// TwinCAT 3 PLC project Cycler
// ProgramVersion: 3.1.4020.4
// libraries:
//   Tc2_Drive, * (Beckhoff Automation GmbH)
//   Tc2_MC2, * (Beckhoff Automation GmbH)
//   Tc2_MC2_Drive, * (Beckhoff Automation GmbH)
//   Tc2_NcDrive, * (Beckhoff Automation GmbH)
//   Tc2_Standard, * (Beckhoff Automation GmbH)
//   Tc2_System, * (Beckhoff Automation GmbH)
//   Tc3_MC2_AdvancedHoming, * (Beckhoff Automation GmbH)
//   Tc3_Module, * (Beckhoff Automation GmbH)
//   VisuDialogs, * (System)
// project tree:
//   DUTs/ AxisInfo.TcDUT, ShutterSide.TcDUT, ShutterState.TcDUT
//   / GlobalTextList.TcGTLO, PlcTask.TcTTO, Visualization Manager.TcVMO (not stored)
//   GVLs/ GVL.TcGVL
//   POUs/ Cycler.TcPOU, TestMotion.TcPOU, MAIN.TcPOU
//   VISUs/ CyclerGUI.TcVIS, TestMotionGUI.TcVIS
// real-time tasks:
//   TASK PlcTask: cycle T#1ms, priority 20, ADS port 350
// motion (NC):
//   TASK NC-Task 1 SAF: cycle T#1ms, priority 4, ADS port 501
//   TASK NC-Task 1 SVB: cycle T#10ms, priority 8, ADS port 511
//   AXIS Axis 1 (id 1)
//     Dynamic: Acceleration=7407.41, Deceleration=7407.41, Jerk=32921.8
//     Velo: RefSearch=60, SlowManual=150
//     OtherSettings: AllowMotionCmdToSlave=true
//     encoder EncType=4
//       EncPara: ScaleFactorNumerator=0.049777676567, MaxCount=#x0000ffff
//         SoftEndMaxControl: Range=749
//         Inc: RefSearchInverse=true, RefSyncInverse=false, RefSoftSyncMask=#x0000ffff
//         TimeComp: TimeCompMode=1, EncDelayCycles=4
//     drive DrvType=24
//       Analog: VeloReferenz=2038.894
//       TimeComp: TaskDelayCycles=1
//     controller CtrType=1
//       CtrPara: PriorControlFactor=1
//         PosDiffControl: Range=2.5, Time=0.01
//         Observer: BandWidth=20
//   AXIS Axis 2 (id 2)
//     Dynamic: Acceleration=7407.41, Deceleration=7407.41, Jerk=32921.8
//     Velo: RefSearch=60
//     OtherSettings: AllowMotionCmdToSlave=true
//     encoder EncType=4
//       EncPara: ScaleFactorNumerator=0.049777676567, MaxCount=#x0000ffff
//         SoftEndMaxControl: Range=749
//         Inc: RefSoftSyncMask=#x0000ffff
//         TimeComp: TimeCompMode=1, EncDelayCycles=4
//     drive DrvType=24
//       Analog: VeloReferenz=2038.894
//       TimeComp: TaskDelayCycles=1
//     controller CtrType=1
//       CtrPara: PriorControlFactor=1
//         PosDiffControl: Range=2.5, Time=0.01
//         Observer: BandWidth=20
// I/O:
//   DEVICE Device 1 (EtherCAT), AmsNetId 5.48.66.18.2.1
//     Term 1 (EK1200) [EK1200-5000 EtherCAT Power supply (2A E-Bus)]
//       Term 2 (EL7047) [EL7047 1Ch. Stepper motor output stage (50V, 5A)]
//       Term 3 (EL1819) [EL1819 16Ch. Dig. Input 24V, 10µs]
//       Term 9 (EL1258) [EL1258 8Ch. Dig Input 24V with Multi-Time-Stamp]
//       Term 10 (EL1259) [EL1259 8Ch. Dig Input 24V/8Ch. Dig. Output 24V with Multi-Time-Stamp]
//       Term 4 (EL7047) [EL7047 1Ch. Stepper motor output stage (50V, 5A)]
//       Term 5 (EL2622) [EL2622 2Ch. Relay Output, NO (230V AC / 30V DC)]
//       Term 14 (EK1110) [EK1110 EtherCAT extension]
//     Term 15 (EK1100) [EK1100 EtherCAT Coupler (2A E-Bus)]
//       Term 16 (EL3681) [EL3681 Digital multimeter terminal]
//       Term 17 (EL3318) [EL3318 8Ch. Ana Input Thermocouple (TC)]
//       Term 23 (EL9011) [EL9011 End Terminal]
//     Term 18 (EK1100) [EK1100 EtherCAT Coupler (2A E-Bus)]
//       Term 19 (EL3602) [EL3602 2Ch. Ana. Input +/-10Volt, Diff. 24bit]
//       Term 20 (EL3602) [EL3602 2Ch. Ana. Input +/-10Volt, Diff. 24bit]
//       Term 24 (EL9011) [EL9011 End Terminal]
// variable links:
//   (this object) <-> Device 1 (EtherCAT)/Term 1 (EK1200)/Term 2 (EL7047)
//     Drive/Inputs/In/nState1 @bit 3 <-> STM Status/Status/Error
//     Drive/Inputs/In/nState1 @bit 7 <-> STM Status/Status/Motor stall
//     Drive/Inputs/In/nState1 @bit 5 <-> STM Status/Status/Moving negative
//     Drive/Inputs/In/nState1 @bit 4 <-> STM Status/Status/Moving positive
//     Drive/Inputs/In/nState1 @bit 1 <-> STM Status/Status/Ready
//     Drive/Inputs/In/nState1 <-> STM Status/Status/Ready to enable
//     Drive/Inputs/In/nState1 @bit 6 <-> STM Status/Status/Torque reduced
//     Drive/Inputs/In/nState1 @bit 2 <-> STM Status/Status/Warning
//     Drive/Inputs/In/nState2 @bit 4 <-> STM Status/Status/Digital input 2
//     Drive/Inputs/In/nState2 @bit 5 <-> STM Status/Status/Sync error
//     Drive/Inputs/In/nState2 @bit 7 <-> STM Status/Status/TxPDO Toggle
//     Drive/Inputs/In/nState4 @bit 1 <-> WcState/InputToggle
//     Drive/Inputs/In/nState4 <-> WcState/WcState
//     Drive/Outputs/Out/nCtrl1 <-> STM Control/Control/Enable
//     Drive/Outputs/Out/nCtrl1 @bit 2 <-> STM Control/Control/Reduce torque
//     Drive/Outputs/Out/nCtrl1 @bit 1 <-> STM Control/Control/Reset
//     Drive/Outputs/Out/nCtrl2 @bit 3 <-> STM Control/Control/Digital output 1
//     Drive/Outputs/Out/nDataOut2[0] <-> STM Velocity/Velocity
//     Enc/Inputs/In/nDataIn1[0] <-> ENC Status compact/Counter value
//     Enc/Inputs/In/nDataIn2[0] <-> ENC Status compact/Latch value
//     Enc/Inputs/In/nState1 @bit 4 <-> ENC Status compact/Status/Counter overflow
//     Enc/Inputs/In/nState1 @bit 3 <-> ENC Status compact/Status/Counter underflow
//     Enc/Inputs/In/nState1 @bit 7 <-> ENC Status compact/Status/Extrapolation stall
//     Enc/Inputs/In/nState1 <-> ENC Status compact/Status/Latch C valid
//     Enc/Inputs/In/nState1 @bit 1 <-> ENC Status compact/Status/Latch extern valid
//     Enc/Inputs/In/nState1 @bit 2 <-> ENC Status compact/Status/Set counter done
//     Enc/Inputs/In/nState2 @bit 4 <-> ENC Status compact/Status/Status of extern latch
//     Enc/Inputs/In/nState2 <-> ENC Status compact/Status/Status of input A
//     Enc/Inputs/In/nState2 @bit 1 <-> ENC Status compact/Status/Status of input B
//     Enc/Inputs/In/nState2 @bit 2 <-> ENC Status compact/Status/Status of input C
//     Enc/Inputs/In/nState2 @bit 5 <-> ENC Status compact/Status/Sync error
//     Enc/Inputs/In/nState2 @bit 7 <-> ENC Status compact/Status/TxPDO Toggle
//     Enc/Inputs/In/nState4 @bit 1 <-> WcState/InputToggle
//     Enc/Inputs/In/nState4 <-> WcState/WcState
//     Enc/Outputs/Out/nCtrl1 <-> ENC Control compact/Control/Enable latch C
//     Enc/Outputs/Out/nCtrl1 @bit 3 <-> ENC Control compact/Control/Enable latch extern on negative edge
//     Enc/Outputs/Out/nCtrl1 @bit 1 <-> ENC Control compact/Control/Enable latch extern on positive edge
//     Enc/Outputs/Out/nCtrl1 @bit 2 <-> ENC Control compact/Control/Set counter
//     Enc/Outputs/Out/nDataOut1[0] <-> ENC Control compact/Set counter value
//   (this object) <-> Device 1 (EtherCAT)/Term 1 (EK1200)/Term 4 (EL7047)
//     Drive/Inputs/In/nState1 @bit 3 <-> STM Status/Status/Error
//     Drive/Inputs/In/nState1 @bit 7 <-> STM Status/Status/Motor stall
//     Drive/Inputs/In/nState1 @bit 5 <-> STM Status/Status/Moving negative
//     Drive/Inputs/In/nState1 @bit 4 <-> STM Status/Status/Moving positive
//     Drive/Inputs/In/nState1 @bit 1 <-> STM Status/Status/Ready
//     Drive/Inputs/In/nState1 <-> STM Status/Status/Ready to enable
//     Drive/Inputs/In/nState1 @bit 6 <-> STM Status/Status/Torque reduced
//     Drive/Inputs/In/nState1 @bit 2 <-> STM Status/Status/Warning
//     Drive/Inputs/In/nState2 @bit 4 <-> STM Status/Status/Digital input 2
//     Drive/Inputs/In/nState2 @bit 5 <-> STM Status/Status/Sync error
//     Drive/Inputs/In/nState2 @bit 7 <-> STM Status/Status/TxPDO Toggle
//     Drive/Inputs/In/nState4 @bit 1 <-> WcState/InputToggle
//     Drive/Inputs/In/nState4 <-> WcState/WcState
//     Drive/Outputs/Out/nCtrl1 <-> STM Control/Control/Enable
//     Drive/Outputs/Out/nCtrl1 @bit 2 <-> STM Control/Control/Reduce torque
//     Drive/Outputs/Out/nCtrl1 @bit 1 <-> STM Control/Control/Reset
//     Drive/Outputs/Out/nCtrl2 @bit 3 <-> STM Control/Control/Digital output 1
//     Drive/Outputs/Out/nDataOut2[0] <-> STM Velocity/Velocity
//     Enc/Inputs/In/nDataIn1[0] <-> ENC Status compact/Counter value
//     Enc/Inputs/In/nDataIn2[0] <-> ENC Status compact/Latch value
//     Enc/Inputs/In/nState1 @bit 4 <-> ENC Status compact/Status/Counter overflow
//     Enc/Inputs/In/nState1 @bit 3 <-> ENC Status compact/Status/Counter underflow
//     Enc/Inputs/In/nState1 @bit 7 <-> ENC Status compact/Status/Extrapolation stall
//     Enc/Inputs/In/nState1 <-> ENC Status compact/Status/Latch C valid
//     Enc/Inputs/In/nState1 @bit 1 <-> ENC Status compact/Status/Latch extern valid
//     Enc/Inputs/In/nState1 @bit 2 <-> ENC Status compact/Status/Set counter done
//     Enc/Inputs/In/nState2 @bit 4 <-> ENC Status compact/Status/Status of extern latch
//     Enc/Inputs/In/nState2 <-> ENC Status compact/Status/Status of input A
//     Enc/Inputs/In/nState2 @bit 1 <-> ENC Status compact/Status/Status of input B
//     Enc/Inputs/In/nState2 @bit 2 <-> ENC Status compact/Status/Status of input C
//     Enc/Inputs/In/nState2 @bit 5 <-> ENC Status compact/Status/Sync error
//     Enc/Inputs/In/nState2 @bit 7 <-> ENC Status compact/Status/TxPDO Toggle
//     Enc/Inputs/In/nState4 @bit 1 <-> WcState/InputToggle
//     Enc/Inputs/In/nState4 <-> WcState/WcState
//     Enc/Outputs/Out/nCtrl1 <-> ENC Control compact/Control/Enable latch C
//     Enc/Outputs/Out/nCtrl1 @bit 3 <-> ENC Control compact/Control/Enable latch extern on negative edge
//     Enc/Outputs/Out/nCtrl1 @bit 1 <-> ENC Control compact/Control/Enable latch extern on positive edge
//     Enc/Outputs/Out/nCtrl1 @bit 2 <-> ENC Control compact/Control/Set counter
//     Enc/Outputs/Out/nDataOut1[0] <-> ENC Control compact/Set counter value
//   Cycler Instance <-> Device 1 (EtherCAT)/Term 1 (EK1200)/Term 2 (EL7047)
//     PlcTask Inputs/GVL.limitHomeXp <-> STM Status/Status/Digital input 1
//   Cycler Instance <-> Device 1 (EtherCAT)/Term 1 (EK1200)/Term 4 (EL7047)
//     PlcTask Inputs/GVL.limitHomeXm <-> STM Status/Status/Digital input 1
//   Cycler Instance <-> Device 1 (EtherCAT)/Term 1 (EK1200)/Term 5 (EL2622)
//     PlcTask Outputs/GVL.brakeRelays <-> Channel 1/Output
//     PlcTask Outputs/GVL.brakeRelays <-> Channel 2/Output
//   Cycler Instance <-> NC-Task 1 SAF/Axes/Axis 1
//     PlcTask Inputs/MAIN.physicalAxes[0].NcToPlc <-> Outputs/ToPlc
//     PlcTask Outputs/MAIN.physicalAxes[0].PlcToNc <-> Inputs/FromPlc
//   Cycler Instance <-> NC-Task 1 SAF/Axes/Axis 2
//     PlcTask Inputs/MAIN.physicalAxes[1].NcToPlc <-> Outputs/ToPlc
//     PlcTask Outputs/MAIN.physicalAxes[1].PlcToNc <-> Inputs/FromPlc

CONFIGURATION Cycler
    RESOURCE PLC ON TwinCAT3
        TASK PlcTask(INTERVAL := T#1ms, PRIORITY := 20);
        PROGRAM MAIN WITH PlcTask : MAIN;
    END_RESOURCE
END_CONFIGURATION

// ---- DUTs/AxisInfo.TcDUT
TYPE AxisInfo :
STRUCT
	openPosition: LREAL;
	closedPosition: LREAL;
END_STRUCT
END_TYPE

// ---- DUTs/ShutterSide.TcDUT
{attribute 'qualified_only'}
(****************** {attribute 'strict'} *)(* Want to treat them as integer constants*)
TYPE ShutterSide :
(
	MINUSX, (* The -X side.*)
    PLUSX   (* The +X side.*)
)INT;
END_TYPE

// ---- DUTs/ShutterState.TcDUT
{attribute 'qualified_only'}
{attribute 'strict'}
TYPE ShutterState :
(
	STOPPED,    (* No motion, positions indeterminate. *)
	RESETTING,  (* No motion, clearing axis faults. *)
	ENABLING,   (* No motion, re-enabling axes after a reset. *)
	OPENING,    (* One blade set is retracting, the other is still. *)
	CLOSING,    (* One blade set is extending, the other is still. *)
	CLOSED      (* One blade set is fully retracted, the other is fully extended. *)
);
END_TYPE

// ---- GVLs/GVL.TcGVL
{attribute 'qualified_only'}
VAR_GLOBAL
	task						: 	INT 	:= 0;
	brakeRelays 		AT %Q*	:	BYTE;

	
	//Home and deployed switches
	limitHomeXp 	AT %I*	: 	BOOL;
	limitDeployedXp	AT %I*	: 	BOOL;
	limitHomeXm 	AT %I*	: 	BOOL;
	limitDeployedXm	AT %I*	: 	BOOL;
END_VAR

// ---- POUs/MAIN.TcPOU
PROGRAM MAIN
VAR
	cycler		: Cycler;
	physicalAxes: ARRAY [ShutterSide.PLUSX .. ShutterSide.MINUSX] OF AXIS_REF; (* Must be linked to Axis1 and 2, respectively, under MOTION. *)
	axisInfo	: ARRAY [ShutterSide.PLUSX..SHutterSide.MINUSX] OF AxisInfo := [(openPosition:=0.0, closedPosition:=749.0), (openPosition:=749.0, closedPosition:=0.0)];
	start, stop, reset, abort: BOOL;
	delay		: TON;
	acceleration, speed: LREAL;
	exposure	: TIME;
	

	testMotion		: TestMotion;
	home 			: BYTE;
	testMotionState	: INT :=100;
	nextInstruct	: BOOL;
END_VAR
VAR CONSTANT
	accTitle	: STRING := 'Acceleration';
END_VAR

delay(IN:=TRUE, PT:=T#0S);
IF speed>1666 THEN 
	speed:=0;
END_IF
IF delay.Q THEN
    delay(IN:=FALSE);
	
	CASE GVL.task OF
		1:
		cycler(
        	physicalAxes	:= physicalAxes,
        	axisInfo 		:= axisInfo,
        	abortRequest	:= abort,
        	resetRequest	:= reset,
        	startRequest	:= start,
        	stopRequest		:= stop,
        	exposureTime	:= exposure,
        	speed			:= speed,
        	acceleration	:= acceleration);
			
		2:
		testMotion(
			axisXP 			:= physicalAxes[ShutterSide.PLUSX],
			axisXM 			:= physicalAxes[ShutterSide.MINUSX],
			abortRequest	:= abort,
        	resetRequest	:= reset,
        	startRequest	:= start,
        	stopRequest		:= stop,
			homeRequest		:= home,
			speed			:= speed,
			state			:= testMotionState,
			nextInstruct	:= nextInstruct);

	END_CASE



END_IF

END_PROGRAM

// ---- POUs/Cycler.TcPOU
FUNCTION_BLOCK PUBLIC Cycler
VAR_IN_OUT
	physicalAxes: ARRAY [ShutterSide.MINUSX .. ShutterSide.PLUSX] OF AXIS_REF;
	abortRequest, resetRequest, startRequest, stopRequest: BOOL;
END_VAR
VAR_INPUT
	axisInfo: ARRAY [ShutterSide.MINUSX .. ShutterSide.PLUSX] OF AxisInfo;
	speed, acceleration: LREAL;
	exposureTime: TIME;
END_VAR
VAR_OUTPUT
	state: ShutterState := ShutterState.STOPPED;
END_VAR

VAR
	retracting: ShutterSide;
	extending: ShutterSide;
	retractor, extender: MC_MoveAbsolute;
	plusResetter, minusResetter: MC_Reset;
	plusEnabler, minusEnabler: MC_Power;
	expoTimer: TON;
	axisError: ARRAY [ShutterSide.MINUSX .. ShutterSide.PLUSX] OF UDINT;
	brakeRelays AT %Q*: BYTE;	
END_VAR
VAR CONSTANT
	BRAKES_OFF: BYTE := 3;
	BRAKES_ON:  BYTE := 0;
END_VAR


CASE state OF
	ShutterState.STOPPED:
	plusResetter(Axis:=physicalAxes[ShutterSide.PLUSX], Execute:=FALSE);
	minusResetter(Axis:=physicalAxes[ShutterSide.MINUSX], Execute:=FALSE);
	extender(Execute:=FALSE, Axis:=physicalAxes[ShutterSide.PLUSX]);
	retractor(Execute:=FALSE, Axis:=physicalAxes[ShutterSide.MINUSX]);
	expoTimer(IN:=FALSE);
	IF resetRequest THEN
		resetRequest := FALSE;
		state := ShutterState.RESETTING;
	ELSIF startRequest THEN
		startRequest := FALSE;
		retracting :=  ShutterSide.MINUSX;
		extending := ShutterSide.PLUSX;
		state := ShutterState.OPENING;
		brakeRelays := BRAKES_OFF;
	END_IF
	
	ShutterState.OPENING:
	retractor(Axis:=physicalAxes[retracting],
        Execute:=TRUE,
        Position:=axisInfo[retracting].openPosition,
        Velocity:=speed,
        Acceleration:=acceleration,
        Deceleration:=acceleration);
	IF retractor.Error OR retractor.CommandAborted THEN
		state := ShutterState.STOPPED;
		brakeRelays := BRAKES_ON;
		retractor(Axis:=physicalAxes[retracting], Execute:=FALSE);
		axisError[retracting] := retractor.ErrorID;		
	END_IF
	(* The exposure starts when the first blade set starts to retract. If the blade
       set doesn't reach its target by the time the exposure is supposed to
       be over then the exposure will be extended until it motion is completed.
    *)
	expoTimer(IN:=TRUE, PT:=exposureTime);
	IF expoTimer.Q  AND retractor.Done THEN
		expoTimer(IN:=FALSE);
		retractor(Axis:=physicalAxes[retracting], Execute:=FALSE);
		state := ShutterState.CLOSING;
	END_IF
	
	ShutterState.CLOSING:
	extender(Axis:=physicalAxes[extending],
        Execute:=TRUE,
        Position:=axisInfo[extending].closedPosition,
        Velocity:=speed,
        Acceleration:=acceleration,
        Deceleration:=acceleration);
	IF extender.Error OR extender.CommandAborted THEN
		state := ShutterState.STOPPED;
		brakeRelays := BRAKES_ON;
		extender(Axis:=physicalAxes[extending], Execute:=FALSE);
		axisError[extending] := extender.ErrorID;
	ELSIF extender.Done THEN
		extender(Axis:=physicalAxes[extending], Execute:=FALSE);
		state := ShutterState.CLOSED;
	END_IF
	
	ShutterState.CLOSED:
	state := ShutterState.OPENING;
	(* Sides now exchange roles. *)
	retracting := ShutterSide.PLUSX - retracting;
	extending := ShutterSide.PLUSX - extending;
	IF stopRequest THEN
		stopRequest := FALSE;
		state := ShutterState.STOPPED;
		brakeRelays := BRAKES_ON;
	END_IF
	
	ShutterState.RESETTING:
	plusResetter(Axis:=physicalAxes[ShutterSide.PLUSX],
        Execute:=TRUE,
        ErrorID => axisError[ShutterSide.PLUSX]);
	minusResetter(Axis:=physicalAxes[ShutterSide.MINUSX],
		Execute:=TRUE,
		ErrorID => axisError[ShutterSide.MINUSX]);
	IF (plusResetter.Done OR plusResetter.Error) AND (minusResetter.Done OR minusResetter.Error) THEN
		IF plusResetter.Done AND minusResetter.Done THEN
	        state := ShutterState.ENABLING;
		ELSE
			state := ShutterState.STOPPED;
			brakeRelays := BRAKES_ON;
		END_IF
	END_IF
	
	ShutterState.ENABLING:
	plusResetter(Axis:=physicalAxes[ShutterSide.PLUSX], Execute:=FALSE);
	minusResetter(Axis:=physicalAxes[ShutterSide.MINUSX], Execute:=FALSE);
	plusEnabler(Axis:=physicalAxes[ShutterSide.PLUSX],
		Enable:=TRUE,
        Enable_Positive:=TRUE,
		Enable_Negative:=TRUE,
		Override:=100.0,
		ErrorID => axisError[ShutterSide.PLUSX]
        );
	minusEnabler(Axis:=physicalAxes[ShutterSide.MINUSX],
        Enable:=TRUE,
        Enable_Positive:=TRUE,
        Enable_Negative:=TRUE,
        Override:=100.0,
        ErrorID => axisError[ShutterSide.MINUSX]);
	IF (plusEnabler.Status OR plusEnabler.Error) AND (minusEnabler.Status OR minusEnabler.Error) THEN
	    state := ShutterState.STOPPED;
		brakeRelays := BRAKES_ON;
	END_IF
	ELSE
		abortRequest := TRUE;
END_CASE
IF abortRequest THEN
	abortRequest := FALSE;
	plusEnabler(Axis:=physicalAxes[ShutterSide.PLUSX], Enable:=FALSE);
	minusEnabler(Axis:=physicalAxes[ShutterSide.MINUSX], Enable:=FALSE);
	state := ShutterState.STOPPED;
	brakeRelays := BRAKES_ON;
END_IF

END_FUNCTION_BLOCK

// ---- POUs/TestMotion.TcPOU
FUNCTION_BLOCK TestMotion
VAR_IN_OUT
	axisXP  : AXIS_REF; //Axis 1;
	axisXM : AXIS_REF; //Axis 2;
	nextInstruct, abortRequest, resetRequest, startRequest, stopRequest: BOOL;
	homeRequest : BYTE;
		
	//statemachine
	state : INT;
	
END_VAR
VAR_INPUT

	speed : LREAL;	

END_VAR
VAR_OUTPUT
END_VAR
VAR
	//test variable
	xPlusMoving : BOOL;
	xMinusMoving : BOOL;
	
	//power 
	mcPowerXP : MC_Power;
	mcPowerXM : MC_Power;
	mcResetXP : MC_Reset;
	mcResetXM : MC_Reset;
	
	//motion
	mcMoveAbsXP : MC_MoveAbsolute;
	mcMoveAbsXM : MC_MoveAbsolute;
	mcHomeXP 	: MC_Home;
	mcHomeXM 	: MC_Home;
	mcHalt		: MC_Halt;
	
	//position
	mcSetPosXP : MC_SetPosition;
	mcSetPosXM : MC_SetPosition;
	
	//error var
	errorIDXP : UDINT;
	errorIDXM : UDINT;
	
END_VAR
VAR CONSTANT
	BRAKES_OFF_C	: BYTE	:= 3;
	BRAKES_ON_C		: BYTE	:= 0;
	HOME_VEL_C		: LREAL	:= 30;
	POSITION_VEL_C	: LREAL := 300;
	POS_START_C		: LREAL := 0;
	POS_END_C		: LREAL := 749;
	HOMEOFFSET_XP_C	: LREAL	:= (POS_START_C+35);
	HOMEOFFSET_XM_C	: LREAL	:= (POS_END_C-88);
END_VAR


axisXP.ReadStatus();
axisXM.ReadStatus();
xPlusMoving  := axisXP.Status.Moving;
xMinusMoving := axisXM.Status.Moving;

//reset input from GUI
IF abortRequest THEN
	abortRequest := FALSE;
	state := -1; //stop state
END_IF
IF resetRequest THEN
	resetRequest := FALSE;
	state := 0;
END_IF

//Homing selection block
IF homeRequest=1 THEN
	state := 200;
ELSIF homeRequest=2 THEN
	state := 300;
ELSIF homeRequest=3 THEN
	state := 400;
END_IF
homeRequest := 0;

//if brakes are not disengaged, disable axis movement
IF GVL.brakeRelays <> 3 THEN
	McPowerXP(Axis := axisXP, Enable := TRUE, Enable_Positive := FALSE, Enable_Negative := FALSE);
	McPowerXM(Axis := axisXM, Enable := TRUE, Enable_Positive := FALSE, Enable_Negative := FALSE);
ELSE
	McPowerXP(Axis := axisXP, Enable := TRUE, Enable_Positive := TRUE, Enable_Negative := TRUE);
	McPowerXM(Axis := axisXM, Enable := TRUE, Enable_Positive := TRUE, Enable_Negative := TRUE); 
END_IF

//if any of the axis is not homed, disable other movement state until homed
IF state>420 THEN
	IF NOT axisXP.Status.Homed OR NOT axisXM.Status.Homed THEN
		abortRequest:=TRUE;
	END_IF
END_IF

CASE state OF
	-1: //Abort state. Disable movement
		McPowerXP(Axis := axisXP, Enable := TRUE, Enable_Positive := FALSE, Enable_Negative := FALSE);
		McPowerXM(Axis := axisXM, Enable := TRUE, Enable_Positive := FALSE, Enable_Negative := FALSE);
		nextInstruct := FALSE;
		GVL.brakeRelays := BRAKES_ON_C;
		
	0: //reset state
		nextInstruct := FALSE;
		mcResetXP(Axis := axisXP, Execute := TRUE, ErrorID => errorIDXP);
		mcResetXM(Axis := axisXM, Execute := TRUE, ErrorID => errorIDXM);
		IF mcResetXP.Error OR mcResetXM.Error THEN
			McPowerXP(Axis := axisXP, Enable := TRUE, Enable_Positive := FALSE, Enable_Negative := FALSE);
			McPowerXM(Axis := axisXM, Enable := TRUE, Enable_Positive := FALSE, Enable_Negative := FALSE);
			GVL.brakeRelays := BRAKES_ON_C;
			state 			:= 100; //go to stop state
		ELSIF mcResetXP.Done AND mcResetXM.Done THEN
			McPowerXP(Axis := axisXP, Enable := TRUE, Enable_Positive := TRUE, Enable_Negative := TRUE);
			McPowerXM(Axis := axisXM, Enable := TRUE, Enable_Positive := TRUE, Enable_Negative := TRUE);
			mcResetXP(Axis := axisXP, Execute := FALSE);
			mcResetXM(Axis := axisXM, Execute := FALSE);
			GVL.brakeRelays	:= BRAKES_OFF_C;
			state 			:= 100; //go to stop state
		END_IF
		
	100: //stop state
		mcMoveAbsXP(Axis := axisXP, Execute := FALSE);
		mcMoveAbsXM(Axis := axisXM, Execute := FALSE);
		mcHomeXP(Axis := axisXP, Execute := FALSE);
		mcHomeXM(Axis := axisXP, Execute := FALSE);
	
		
	200://Homing start for AxisXP
		mcHomeXP(Axis := axisXP, Position := POS_START_C, bCalibrationCam := GVL.limitHomeXp, Execute := TRUE);
		IF mcHomeXP.Done THEN
			state := 210;
		END_IF
		
	210: //Homing routine running for AxisXP
		IF NOT mcHomeXP.Error THEN
			mcHomeXP(Axis := axisXP, Execute := FALSE);
			mcMoveAbsXP(Axis:=axisXP, Execute:= TRUE, Velocity:=HOME_VEL_C, Position:=HOMEOFFSET_XP_C);
			IF mcMoveAbsXP.Done THEN
				mcMoveAbsXP(Axis:=axisXP, Execute:= FALSE);
				mcSetPosXP(Axis:=axisXP, Position:=POS_START_C, Execute:=TRUE);
				state := 220; 
			END_IF
		ELSE
			state :=100; //stop state. Should go to error state
		END_IF
		
	220: //Homing routine complete for AxisXP
		mcSetPosXP(Axis:=axisXP, Execute:=FALSE);
		IF  mcSetPosXP.Done THEN
			state := 100;
		END_IF

		
	300://Homing start for AxisXM
		mcHomeXM(Axis := axisXM, Position := POS_START_C, bCalibrationCam := GVL.limitHomeXm, Execute := TRUE);
		IF mcHomeXM.Done THEN
			state := 310;
		END_IF	


	310: //Homing routine running for AxisXM
		IF NOT mcHomeXM.Error THEN
			mcHomeXM(Axis := axisXM, Execute := FALSE);
			mcMoveAbsXM(Axis:=axisXM, Execute:= TRUE, Velocity:=HOME_VEL_C, Position:=HOMEOFFSET_XM_C);
			IF mcMoveAbsXM.Done THEN
				mcMoveAbsXM(Axis:=axisXM, Execute:= FALSE);
				mcSetPosXM(Axis:=axisXM, Position:=POS_END_C, Execute:=TRUE);
				state := 320; 
			END_IF
		ELSE
			state :=100; //stop state. Should go to error state
		END_IF	
		
	320: //Homing routine complete for AxisXM
		mcSetPosXM(Axis:=axisXM, Execute:=FALSE);
		IF  mcSetPosXM.Done THEN
			state := 100;
		END_IF	

	
	400: //Homing start for both blades
		mcHomeXP(Axis := axisXP, Position := HOMEOFFSET_XP_C, bCalibrationCam := GVL.limitHomeXp, Execute := TRUE);
		mcHomeXM(Axis := axisXM, Position := HOMEOFFSET_XM_C, bCalibrationCam := GVL.limitHomeXm, Execute := TRUE);
		IF mcHomeXP.Done AND mcHomeXM.Done THEN
			state := 410;
		END_IF
		
	410: //Homing running for both blades
		IF NOT mcHomeXP.Error AND NOT mcHomeXM.Error THEN
			mcHomeXP(Axis := axisXP, Execute := FALSE);
			mcMoveAbsXP(Axis:=axisXP, Velocity:=HOME_VEL_C, Position:=POS_START_C, Execute:= TRUE,);
			mcHomeXM(Axis := axisXM, Execute := FALSE);
			mcMoveAbsXM(Axis:=axisXM, Velocity:=HOME_VEL_C, Position:=POS_END_C, Execute:= TRUE);
			IF mcMoveAbsXP.Done AND mcMoveAbsXM.Done THEN
				mcMoveAbsXP(Axis:=axisXP, Execute:= FALSE);
				mcMoveAbsXM(Axis:=axisXM, Execute:= FALSE);
				state := 100; 
			END_IF
		ELSE
			state :=100; //stop state. Should go to error state
		END_IF

	420: //Homing routine complete for AxisXM
		mcSetPosXP(Axis:=axisXP, Execute:=FALSE);
		mcSetPosXM(Axis:=axisXM, Execute:=FALSE);
		IF  mcSetPosXP.Done AND mcSetPosXM.Done THEN
			state := 100;
		END_IF	

//States higher than 420 requires HOMING ROUTINE to be run first.


//Basic Motions ---------------------------------------------------------------
	1000: //Open shutter
		mcMoveAbsXP(Axis:=axisXP, Position:= POS_START_C, Velocity:=speed, Execute:=TRUE);
		mcMoveAbsXM(Axis:=axisXM, Position:= POS_END_C, Velocity:=speed, Execute:=TRUE);
		IF mcMoveAbsXP.Done AND mcMoveAbsXM.Done THEN
			state:=100;
		END_IF
		
		
	1100: //Close shutter towards X+ side. AxisXP retracts to its HOME position
		mcMoveAbsXP(Axis:=axisXP, Position:= POS_START_C, Velocity:=speed, Execute:=TRUE);
		IF mcMoveAbsXP.Done THEN
			mcMoveAbsXP(Axis:=axisXP, Execute:=FALSE);
			state:=1110;
		END_IF
		
	1110: //Close shutter towards X+ side. AxisXM extends to its DEPLOYED position 
		mcMoveAbsXM(Axis:=axisXM, Position:= POS_START_C, Velocity:=speed, Execute:=TRUE);
		IF mcMoveAbsXM.Done THEN
			mcMoveAbsXM(Axis:=axisXM, Execute:=FALSE);
			state:=100;	
		END_IF
		
	1200: //Close shutter towards X- side. AxisXM retracts to its HOME position (~750 mm)
		mcMoveAbsXM(Axis:=axisXM, Position:= POS_END_C, Velocity:=speed, Execute:=TRUE);
		IF mcMoveAbsXM.Done THEN
			mcMoveAbsXM(Axis:=axisXM, Execute:=FALSE);
			state:=1210;
		END_IF
		
	1210: //Close shutter towards X- side. AxisXP extends to its DEPLOYED position
		mcMoveAbsXP(Axis:=axisXP, Position:= POS_END_C, Velocity:=speed, Execute:=TRUE);
		IF mcMoveAbsXP.Done THEN
			mcMoveAbsXP(Axis:=axisXP, Execute:=FALSE);
			state:=100;
		END_IF


//Motion for visit----------------------------------------------------------------------------
		
	2000: //Normal Visit. Put both blades in position at 0 mm - Shutter closed
		mcMoveAbsXP(Axis:=axisXP, Position:=POS_START_C, Velocity:=POSITION_VEL_C, Execute:=TRUE);
		mcMoveAbsXM(Axis:=axisXM, Position:=POS_START_C, Velocity:=POSITION_VEL_C, Execute:=TRUE);
		IF mcMoveAbsXP.Done AND mcMoveAbsXM.Done THEN
			mcMoveAbsXP(Axis:=axisXP, Execute:=FALSE);
			mcMoveAbsXM(Axis:=axisXM, Execute:=FALSE);
			state:=2010;
		END_IF
	
	2010: //Normal Visit. Blade in position. Wait for input to continue.
		IF nextInstruct THEN
			nextInstruct:=FALSE;
			state:=2100;
		END_IF
		
	2100: //Normal Visit. Visit 1 sequence - axisXM travels to end of X- side - Shutter open
		mcMoveAbsXM(Axis:=axisXM, Position:=POS_END_C, Velocity:=speed, Execute:=TRUE);
		IF mcMoveAbsXM.Done THEN
			mcMoveAbsXM(Axis:=axisXM, Execute:=FALSE);
			state:=2110;
		END_IF

	2110: //Normal Visit. Visit 1 sequence - axisXP travels to end of X- side - Shutter close
		mcMoveAbsXP(Axis:=axisXP, Position:=POS_END_C, Velocity:=speed, Execute:=TRUE);
		IF mcMoveAbsXP.Done THEN
			mcMoveAbsXP(Axis:=axisXP, Execute:=FALSE);
			state:=2120;
		END_IF
		
	2120: //Normal Visit. Pause at the end of first visit. Wait for input to continue
		IF nextInstruct THEN
			nextInstruct:=FALSE;
			state:=2200;
		END_IF
	
	2200: //Normal Visit. Visit 2 sequence - axisXP travels to X+ side - Shutter open
		mcMoveAbsXP(Axis:=axisXP, Position:=POS_START_C, Velocity:=speed, Execute:=TRUE);
		IF mcMoveAbsXP.Done THEN
			mcMoveAbsXP(Axis:=axisXP, Execute:=FALSE);
			state:=2210;
		END_IF
		
	2210: //Normal Visit. Visit 2 sequence - axisXM travels to X+ side - Shutter close
		mcMoveAbsXM(Axis:=axisXM, Position:=POS_START_C, Velocity:=speed, Execute:=TRUE);
		IF mcMoveAbsXM.Done THEN
			mcMoveAbsXM(Axis:=axisXM, Execute:=FALSE);
			state:=100;
		END_IF
		
	
	
	
END_CASE

END_FUNCTION_BLOCK

// ---- GlobalTextList.TcGTLO
TEXTLIST GlobalTextList
  9 = '%7.1f'
  12 = '%7.4f'
  13 = '%7.4f mm'
  8 = '%8.1f'
  4 = '%s'
  16 = '10'
  30 = '1666.6'
  1 = 'Abort'
  25 = 'AxisXP move to:'
  14 = 'AXIS_1: %7.4f mm'
  15 = 'AXIS_2: %7.4f mm'
  10 = 'Brakes ENGAGE'
  11 = 'Brakes RELEASE'
  28 = 'Close towards X+'
  29 = 'Close towards X-'
  33 = 'Continue'
  17 = 'Cycler Task'
  19 = 'Home'
  22 = 'Home AxisXM'
  21 = 'Home AxisXP'
  23 = 'Home Both'
  34 = 'Home Routine'
  20 = 'home2'
  36 = 'Motion Control'
  32 = 'Normal Visit'
  27 = 'Open Position'
  0 = 'Reset'
  35 = 'sad'
  5 = 'Set acceleration'
  7 = 'Set exposure time'
  6 = 'Set speed'
  26 = 'Set Speed'
  31 = 'Set Velocity'
  38 = 'Set Velocity%7.1f'
  37 = 'Set Velocity: %7.1f'
  2 = 'Start'
  24 = 'State: %s'
  3 = 'Stop'
  18 = 'TestMotion Task'
END_TEXTLIST

// ---- VISUs/CyclerGUI.TcVIS
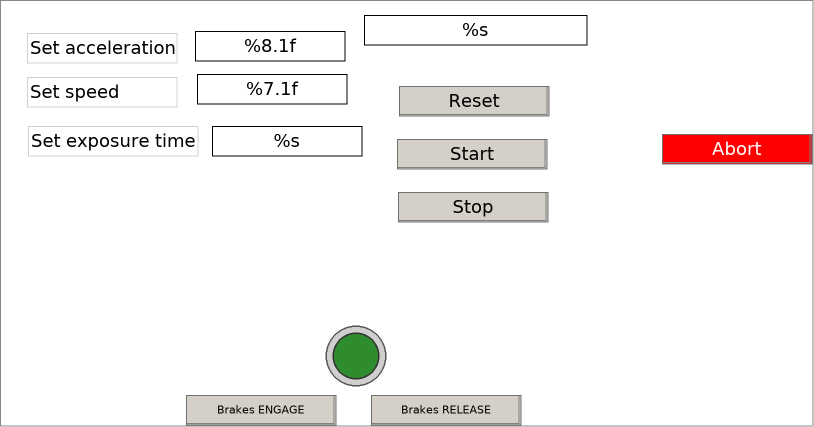
VISUALIZATION CyclerGUI  // 814x427
    Button (399,86 150x30), "Reset", input disabled if: MAIN.cycler.state <> ShutterState.STOPPED
        OnMouseUp: execute { MAIN.reset := TRUE; }
    Button (662,134 150x30), "Abort"
        OnMouseUp: execute { MAIN.abort := TRUE; }
    Button (397,139 150x30), "Start", input disabled if: MAIN.cycler.state <> ShutterState.STOPPED
        OnMouseUp: execute { MAIN.start := TRUE; }
    Button (398,192 150x30), "Stop", input disabled if: MAIN.cycler.state < ShutterState.OPENING
        OnMouseUp: execute { MAIN.stop := TRUE; }
    Rectangle (364,15 223x30), "%s", text variable: MAIN.cycler.state
    Textfield (27,33 150x30), "Set acceleration", input disabled if: MAIN.cycler.state <> ShutterState.STOPPED
        OnMouseUp: write MAIN.acceleration via Default, min 0, max 20000, format %8.1f
    Textfield (27,77 150x30), "Set speed", input disabled if: MAIN.cycler.state <> ShutterState.STOPPED
        OnMouseUp: write MAIN.speed via Default, min 0, max 2000, format %7.1f
    Textfield (28,126 170x30), "Set exposure time", input disabled if: MAIN.cycler.state <> ShutterState.STOPPED
        OnMouseDown: write MAIN.exposure via Default, min T#0s, max T#30s
    Rectangle (195,31 150x30), "%8.1f", text variable: MAIN.acceleration
    Rectangle (197,74 150x30), "%7.1f", text variable: MAIN.speed
    Rectangle (212,126 150x30), "%s", text variable: MAIN.exposure
    Button (186,395 150x30), "Brakes ENGAGE"
        OnMouseClick: execute { MAIN.cycler.brakeRelays := 0; }
    Button (371,395 150x30), "Brakes RELEASE"
        OnMouseClick: execute { MAIN.cycler.brakeRelays := 3; }
    Lamp1 (321,321 70x70), variable: MAIN.cycler.brakeRelays = 3, style: Lamp-Lamp1-Green
END_VISUALIZATION

// ---- VISUs/TestMotionGUI.TcVIS
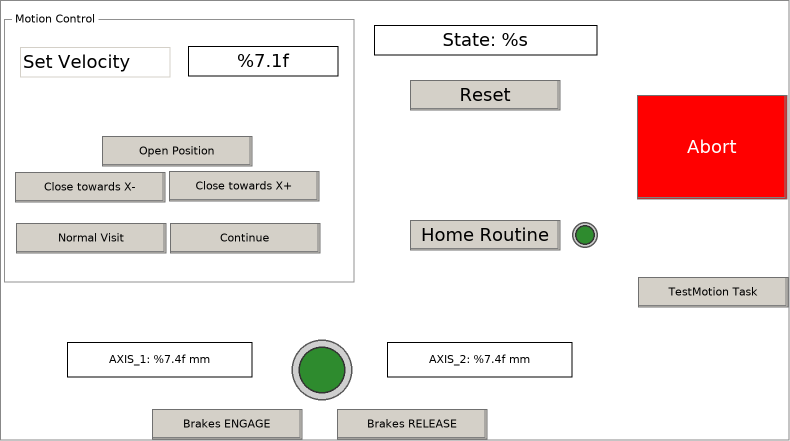
VISUALIZATION TestMotionGUI  // 790x441
    GroupBox (4,11 350x271), "Motion Control"
    Button (152,409 150x30), "Brakes ENGAGE"
        OnMouseClick: execute { GVL.brakeRelays := 0; }
    Button (337,409 150x30), "Brakes RELEASE"
        OnMouseClick: execute { GVL.brakeRelays := 3; }
    Lamp1 (287,335 70x70), variable: GVL.brakeRelays = 3, style: Lamp-Lamp1-Green
    Rectangle (67,342 185x35), "AXIS_1: %7.4f mm", text variable: MAIN.physicalAxes[0].NcToPlc.ActPos
    Rectangle (387,342 185x35), "AXIS_2: %7.4f mm", text variable: MAIN.physicalAxes[1].NcToPlc.ActPos
    Button (638,277 150x30), "TestMotion Task", input disabled if: GVL.task=2;
        OnMouseUp: execute { GVL.task:=2; }
    Button (410,80 150x30), "Reset"
        OnMouseUp: execute { MAIN.reset := TRUE; }
    Button (637,95 150x104), "Abort"
        OnMouseUp: execute { MAIN.abort := TRUE; }
    Rectangle (374,25 223x30), "State: %s", text variable: MAIN.testMotion.state;
    Button (410,220 150x30), "Home Routine", input disabled if: MAIN.testMotion.state <> 100;
        OnMouseUp: execute { MAIN.home := 3; }
    Button (102,136 150x30), "Open Position", input disabled if: MAIN.testMotion.state <> 100;
        OnMouseUp: execute { MAIN.testMotionState:=1000; }
    Textfield (20,47 150x30), "Set Velocity", input disabled if: MAIN.cycler.state <> ShutterState.STOPPED
        OnMouseUp: write MAIN.speed via Default, min 0, max 2000, format %7.1f
    Rectangle (188,46 150x30), "%7.1f", text variable: MAIN.speed
    Button (169,171 150x30), "Close towards X+", input disabled if: MAIN.testMotion.state <> 100;
        OnMouseUp: execute { MAIN.testMotionState:=1100; }
    Button (15,172 150x30), "Close towards X-", input disabled if: MAIN.testMotion.state <> 100;
        OnMouseUp: execute { MAIN.testMotionState:=1200; }
    Button (16,223 150x30), "Normal Visit", input disabled if: MAIN.testMotion.state <> 100;
        OnMouseUp: execute { MAIN.testMotionState:=2000; }
    Button (170,223 150x30), "Continue", input disabled if: MAIN.nextInstruct
        OnMouseUp: execute { MAIN.nextInstruct:=TRUE; }
    Lamp1 (570,220 30x30), variable: MAIN.physicalAxes[0].Status.Homed and MAIN.physicalAxes[1].Status.Homed;, style: Lamp-Lamp1-Green
END_VISUALIZATION
